{attribute 'linkalways'} 
{attribute 'no_explicit_call' := 'This FB is a CLASS and must be accessed using methods or properties'}
{attribute 'enable_dynamic_creation'}
FUNCTION_BLOCK PUBLIC DefaultMoveBuilder IMPLEMENTS I_MoveBuilder, I_MoveAbsoluteBuilder, I_MoveRelativeBuilder
VAR
	_axis : I_Axis;
	_position : LREAL;
	_distance : LREAL;
	_velocity : LREAL;
	_acceleration: LREAL;
	_deceleration: LREAL;
	_jerk: LREAL;
	_bufferMode: AxisBufferMode;
END_VAR

METHOD PUBLIC Acceleration : I_MoveBuilder
VAR_INPUT
	value : LREAL;
END_VAR
_acceleration := value;
Acceleration := THIS^;
END_METHOD

METHOD PUBLIC BufferMode : I_MoveBuilder
VAR_INPUT
	mode : AxisBufferMode;
END_VAR
_bufferMode := mode;
BufferMode := THIS^;
END_METHOD

METHOD PUBLIC BuildMoveAbsoluteCommand : I_MoveCommand
VAR
	pCmd : POINTER TO MoveAbsoluteCommand;
	cmd : I_MoveCommand;
END_VAR
pCmd := __NEW(MoveAbsoluteCommand(
	axis := _axis,
	position := _position,
	velocity := _velocity,
	acceleration := _acceleration,
	deceleration := _deceleration,
	jerk := _jerk,
	bufferMode := _bufferMode
));
BuildMoveAbsoluteCommand := pCmd^;
END_METHOD

METHOD PUBLIC BuildMoveAdditiveCommand : I_MoveCommand
VAR
	pCmd : POINTER TO MoveAdditiveCommand;
	cmd : I_MoveCommand;
END_VAR
pCmd := __NEW(MoveAdditiveCommand(
	axis := _axis,
	distance := _distance,
	velocity := _velocity,
	acceleration := _acceleration,
	deceleration := _deceleration,
	jerk := _jerk,
	bufferMode := _bufferMode
));
BuildMoveAdditiveCommand := pCmd^;
END_METHOD

METHOD PUBLIC BuildMoveRelativeCommand : I_MoveCommand
VAR
	pCmd : POINTER TO MoveRelativeCommand;
	cmd : I_MoveCommand;
END_VAR
pCmd := __NEW(MoveRelativeCommand(
	axis := _axis,
	distance := _distance,
	velocity := _velocity,
	acceleration := _acceleration,
	deceleration := _deceleration,
	jerk := _jerk,
	bufferMode := _bufferMode
));
BuildMoveRelativeCommand := pCmd^;
END_METHOD

METHOD PUBLIC BuildMoveVelocityCommand : I_MoveCommand
VAR
	pCmd : POINTER TO MoveVelocityCommand;
	cmd : I_MoveCommand;
END_VAR
pCmd := __NEW(MoveVelocityCommand(
	axis := _axis,
	velocity := _velocity,
	acceleration := _acceleration,
	deceleration := _deceleration,
	jerk := _jerk,
	bufferMode := _bufferMode
));
BuildMoveVelocityCommand := pCmd^;
END_METHOD

METHOD PUBLIC Deceleration : I_MoveBuilder
VAR_INPUT
	value : LREAL;
END_VAR
_deceleration := value;
Deceleration := THIS^;
END_METHOD

METHOD PUBLIC Distance : I_MoveRelativeBuilder
VAR_INPUT
	value : LREAL;
END_VAR
_distance := value;
Distance := THIS^;
END_METHOD

METHOD FB_init : BOOL
VAR_INPUT
	bInitRetains : BOOL; // if TRUE, the retain variables are initialized (warm start / cold start)
	bInCopyCode : BOOL;  // if TRUE, the instance afterwards gets moved into the copy code (online change)
	axis : I_Axis;
END_VAR
_axis := axis;
END_METHOD

METHOD PUBLIC Jerk : I_MoveBuilder
VAR_INPUT
	value : LREAL;
END_VAR
_jerk := value;
Jerk := THIS^;
END_METHOD

METHOD PUBLIC Position : I_MoveAbsoluteBuilder
VAR_INPUT
	value : LREAL;
END_VAR
_position := value;
Position := THIS^;
END_METHOD

METHOD PUBLIC Velocity : I_MoveBuilder
VAR_INPUT
	value : LREAL;
END_VAR
IF value <= 0 THEN
	_velocity := _axis._InternalParameterSet.fDriveVeloReferenz;
ELSE
	_velocity := value;
END_IF
Velocity := THIS^;
END_METHOD

END_FUNCTION_BLOCK

(* stored: Version 1.1.0.1, ProductVersion 3.1.4024.12
   POU DefaultMoveBuilder: Id {825d4ead-368b-4c60-84d1-d77a39a41a4b}, SpecialFunc None
   Folder Builders: Id {7d62c1e3-7514-4e84-8ffc-b98ce6d2e432}
   Folder Constructor: Id {f807a982-49ba-4dd7-9ec2-e1570a6c97bf}
   Folder Property Setters: Id {b66f7037-2fe6-4aea-b80e-94446af0a964}
   Method Acceleration: Id {ec03430a-e80a-40d9-8e48-b1e12b198d00}
   Method BufferMode: Id {2d0f4c94-0cb5-48e5-a9b3-f44e499ad175}
   Method BuildMoveAbsoluteCommand: Id {733bb99d-343f-41fb-901d-e3a9a3a78c05}
   Method BuildMoveAdditiveCommand: Id {eaf960a2-3fc1-4c11-90ba-254bd777ecf7}
   Method BuildMoveRelativeCommand: Id {9f1a1cda-bbf1-44f3-8b42-fee19e72b447}
   Method BuildMoveVelocityCommand: Id {32bbf258-a34a-4e22-b9e4-d61626652304}
   Method Deceleration: Id {4af86363-85e2-48f2-ab69-3cab5e73f184}
   Method Distance: Id {b263d895-40ab-48e1-a2e9-27af2c754030}
   Method FB_init: Id {49d0d298-9eab-4f96-a580-8b4d3cf67021}
   Method Jerk: Id {37012915-44db-449b-8bc8-74a80b32747a}
   Method Position: Id {232effef-9259-4d37-bb96-1d79aee9e8fe}
   Method Velocity: Id {87a6a725-01c7-40d0-8e57-7a87bc138f34} *)
